PROGRAM FlashBits
VAR_OUTPUT
	Bits : BYTE;
END_VAR
VAR
	MaxFlashFreq	: TIME := T#100MS;
    FlashTimer		: TON;    // timeout timer 
END_VAR

FlashTimer(IN:=NOT FlashTimer.Q,PT:=MaxFlashFreq);
IF FlashTimer.Q THEN
	IF Bits=0 THEN
		Bits :=1;
	ELSE	
		Bits:=Bits+1;
	END_IF
END_IF

END_PROGRAM

(* stored: Version 1.1.0.1, ProductVersion 3.1.4024.10
   POU FlashBits: Id {bf60f8b8-539f-4dd5-b813-9283ee85e8f8}, SpecialFunc None *)
